TYPE RelativeHumidityMeasurementStatuses :
STRUCT
	///Is the relative humidity being measured?
	enabledStatus: EnabledStatus;
	///Is the measurement OK?
	healthStatus: HealthStatus;
	///Alarm status
	alarmStatus: HiHiLoLoAlarmStatus;
END_STRUCT
END_TYPE

(* stored: Version 1.1.0.1, ProductVersion 3.1.4019.2
   DUT RelativeHumidityMeasurementStatuses: Id {817c50be-7de5-4154-9f5a-4e9d5d49c1aa} *)
